{attribute 'OPC.UA.DA.StructuredType' := '1'}
TYPE ST_MixingValveSetParameters :
STRUCT
	nControlModeAlgorithm : E_MixingValveControlMode; //select control mode: position mode, heating mode, cooling mode
	nControlModeManual : E_MixingValveControlMode;
END_STRUCT
END_TYPE

(* stored: Version 1.1.0.1, ProductVersion 3.1.4024.9
   DUT ST_MixingValveSetParameters: Id {53981657-c63e-4e9c-b2a2-389391f1a24f} *)
